// TwinCAT 3 PLC project MAS418_PLC
// ProgramVersion: 3.1.4023.0
// libraries:
//   Tc2_Standard, * (Beckhoff Automation GmbH)
//   Tc2_System, * (Beckhoff Automation GmbH)
//   Tc3_Module, * (Beckhoff Automation GmbH)
//   VisuSymbols,3.5.10.0,System
// project tree:
//   / GlobalTextList.TcGTLO, PlcTask.TcTTO, Visualization Manager.TcVMO (not stored)
//   ControlBox/GVLs/ G_Inputs.TcGVL, G_RealControlBox.TcGVL, G_VB.TcGVL
//   ControlBox/POUs/FunctionBlocks/ FB_ModeRealControlBox.TcPOU, FB_ModeSelector.TcPOU, FB_ModeVisualControlBox.TcPOU (not stored)
//   ControlBox/VISUs/ V_VB.TcVIS
//   Inputs/FunctionBlocks/ FB_AnalogInputScaling.TcPOU, FB_Encoder.TcPOU, FB_FlowMeterInputScaling.TcPOU, FB_JoystickInputScaling.TcPOU
//   Inputs/GVLs/ G_ScaledSensorData.TcGVL, G_RawSensorData.TcGVL
//   Inputs/ P_Inputs.TcPOU
//   Inputs/Structs/ ST_AnalogInput.TcDUT, ST_AnalogInputScaling.TcDUT, ST_AnalogInputStatus.TcDUT, ST_FlowMeterInputScaling.TcDUT, ST_JoystickInputScaling.TcDUT
//   MotionControl/DUTs/ ST_OpenLoopControlCylinderSettings.TcDUT, ST_OpenLoopControlWinchSettings.TcDUT, ST_Parameters.TcDUT, ST_ValveOutput.TcDUT, ST_ValveDeadBand.TcDUT
//   MotionControl/FunctionBlocks/MainBlocks/ FB_ManualControl.TcPOU
//   MotionControl/FunctionBlocks/SubBlocks/ FB_Joystick.TcPOU, FB_OpenLoopCylinderControl.TcPOU, FB_OpenLoopWinchControl.TcPOU, FB_ValveOutput.TcPOU
//   MotionControl/GVLs/ G_Outputs.TcGVL, G_Parameters.TcGVL, G_Work.TcGVL
//   MotionControl/POUs/ P_CraneControl.TcPOU, P_Outputs.TcPOU
//   Programs/ MAIN.TcPOU
//   ControlBox/DUTs/ E_Button.TcDUT (not stored), E_Joy.TcDUT (not stored), E_Light.TcDUT (not stored), E_Mode.TcDUT, E_Status.TcDUT (not stored)
//   ControlBox/Interfaces/ I_ControlType.TcIO, I_Mode.TcIO (not stored)
// real-time tasks:
//   TASK PlcTask: cycle T#10ms, priority 20, ADS port 350
// I/O:
//   DEVICE Device 4 (EtherCAT) (disabled), AmsNetId 5.80.90.242.5.1
//     Term 1 (EK1100) [EK1100 EtherCAT Coupler (2A E-Bus)]
//       Term 2 (EL1008)
//       Term 3 (EL2008)
//       Term 4 (EL3068)
//       Term 5 (EL3068)
//       Term 6 (EL3174) [EL3174 4Ch. Ana. Input +/-10V Diff., +/-20mA SingleEnded, 16 Bit]
//       Term 7 (EL3255)
//       Term 8 (EL4104)
//       Term 10 (EL9011) [EL9011 End Terminal]
//     Box 9 (Fraba EtherCAT) [Absolute Rotary Encoder IXARC V01.05]
// variable links:
//   MAS418-PLC/MAS418-PLC Instance <-> Device 4 (EtherCAT)/Term 1 (EK1100)/Term 2 (EL1008)
//     PlcTask Inputs/G_RawSensorData.bAutoModeSelector <-> Channel 2/Input
//     PlcTask Inputs/G_RawSensorData.bJoystickEnable <-> Channel 5/Input
//     PlcTask Inputs/G_RawSensorData.bManualModeSelector <-> Channel 1/Input
//     PlcTask Inputs/G_RawSensorData.bStartButton <-> Channel 3/Input
//     PlcTask Inputs/G_RawSensorData.bStopButton <-> Channel 4/Input
//   MAS418-PLC/MAS418-PLC Instance <-> Device 4 (EtherCAT)/Term 1 (EK1100)/Term 7 (EL3255)
//     PlcTask Inputs/G_RawSensorData.stJoyX.nValue <-> AI Standard Channel 2/Value
//     PlcTask Inputs/G_RawSensorData.stJoyY.nValue <-> AI Standard Channel 3/Value
//     PlcTask Inputs/G_RawSensorData.stPositionCylinder.nValue <-> AI Standard Channel 1/Value

CONFIGURATION MAS418_PLC
    RESOURCE PLC ON TwinCAT3
        TASK PlcTask(INTERVAL := T#10ms, PRIORITY := 20);
        PROGRAM MAIN WITH PlcTask : MAIN;
    END_RESOURCE
END_CONFIGURATION

// ---- Inputs/Structs/ST_AnalogInput.TcDUT
TYPE ST_AnalogInput :
STRUCT
	stStatus AT %I* : ST_AnalogInputStatus;
	nValue AT %I* : INT;
END_STRUCT
END_TYPE

// ---- Inputs/Structs/ST_AnalogInputScaling.TcDUT
TYPE ST_AnalogInputScaling :
STRUCT
	fMaxInputValue : LREAL;
	fMinInputValue : LREAL;
	fMaxOutputValue : LREAL;
	fMinOutputValue : LREAL;
END_STRUCT
END_TYPE

// ---- Inputs/Structs/ST_AnalogInputStatus.TcDUT
TYPE ST_AnalogInputStatus :
STRUCT
	Underrange : BIT;
	Overrange : BIT;
	Limit_1_0 : BIT;
	Limit_1_1 : BIT;
	Limit_2_0 : BIT;
	Limit_2_1 : BIT;
	Error : BIT;
	Reserved_0_7 : BIT;
	Reserved_1_0 : BIT;	
	Reserved_1_1 : BIT;
	Reserved_1_2 : BIT;	
	Reserved_1_3 : BIT;		
	Reserved_1_4 : BIT;	
	Reserved_1_5 : BIT;	
	TxPDO_State : BIT;
	TxPDO_Toggle : BIT;
END_STRUCT
END_TYPE

// ---- Inputs/Structs/ST_FlowMeterInputScaling.TcDUT
TYPE ST_FlowMeterInputScaling :
STRUCT
	fMaxInputValue : LREAL;
	fMinInputValue : LREAL;
	fNeutralInputValue : LREAL;
	fNeutralDeadband : LREAL;
	fMaxOutputValue : LREAL;
	fMinOutputValue : LREAL;
	fNeutralOutputValue : LREAL;
END_STRUCT
END_TYPE

// ---- Inputs/Structs/ST_JoystickInputScaling.TcDUT
TYPE ST_JoystickInputScaling :
STRUCT
	fMaxInputValue : LREAL;
	fMinInputValue : LREAL;
	fNeutralInputValue : LREAL;
	fNeutralDeadband : LREAL;
	fMaxOutputValue : LREAL;
	fMinOutputValue : LREAL;
	fNeutralOutputValue : LREAL;
END_STRUCT
END_TYPE

// ---- MotionControl/DUTs/ST_OpenLoopControlCylinderSettings.TcDUT
TYPE ST_OpenLoopControlCylinderSettings :
STRUCT
	fBoreArea : LREAL := 0.0033183;
	fAnnulusArea : LREAL := 0.0023562;
	fMaxFlowCapacity : LREAL := 75;
END_STRUCT
END_TYPE

// ---- MotionControl/DUTs/ST_OpenLoopControlWinchSettings.TcDUT
TYPE ST_OpenLoopControlWinchSettings :
STRUCT
	fWichDrumDiameter : LREAL := 0.0475;
	fWinchDisplacement : LREAL := 32;
	fGearBox : LREAL := 20;
	fMaxFlow : LREAL := 60;
	fWinchDrumScaling : LREAL := 0.000744309;
END_STRUCT
END_TYPE

// ---- MotionControl/DUTs/ST_Parameters.TcDUT
TYPE ST_Parameters :
STRUCT
	fCyclicTime : LREAL := 0.01;
	fMaxVelocityLimit : LREAL := 0.05;
	stOpenLoopControlCylinderSettings : ST_OpenLoopControlCylinderSettings;
	stOpenLoopControlWinchSettings : ST_OpenLoopControlWinchSettings;
	fEncoderOffset : LREAL := 17574.8; 
	bDeadBandCompOn : BOOL := TRUE;
	stWinchValveDeadBand : ST_ValveDeadBand := (fPosMax := 29490.0, fPosMin := 20950.0, fNegMin := 18250.0, fNegMax := 9830.0);
	stCylValveDeadBand 	: ST_ValveDeadBand := (fPosMax := 29490.0, fPosMin := 20950.0, fNegMin := 18250.0, fNegMax := 9830.0);
	stJoystickInputScalingY	: ST_JoystickInputScaling := (fMaxInputValue := 20509.0, fMinInputValue := 11787.0, fNeutralInputValue := 16175, fNeutralDeadband := 50.0, fMaxOutputValue := 1.0, fMinOutputValue := -1.0, fNeutralOutputValue := 0.0);
	stJoystickInputScalingX	: ST_JoystickInputScaling := (fMaxInputValue := 20509.0, fMinInputValue := 11787.0, fNeutralInputValue := 16175, fNeutralDeadband := 50.0, fMaxOutputValue := 1.0, fMinOutputValue := -1.0, fNeutralOutputValue := 0.0);
	stCylPistonPositionScaling : ST_AnalogInputScaling := (fMaxInputValue := 32295.0, fMinInputValue := 229.0, fMaxOutputValue := 0.5, fMinOutputValue := 0.0);
	stPressureSensorScaling400bar : ST_AnalogInputScaling := (fMaxInputValue := 32767.0, fMinInputValue := 0.0, fMaxOutputValue := 400.0, fMinOutputValue := 0.0);
	stPressureSensorScaling40bar : ST_AnalogInputScaling := (fMaxInputValue := 32767.0, fMinInputValue := 0.0, fMaxOutputValue := 40.0, fMinOutputValue := 0.0);
	stFlowMeterInputScaling : ST_FlowMeterInputScaling := (fMaxInputValue := 32295.0, fMinInputValue := 0.0, fNeutralInputValue := 15450, fNeutralDeadband := 50.0, fMaxOutputValue := 150.0, fMinOutputValue := -150.0, fNeutralOutputValue := 0.0);
END_STRUCT
END_TYPE

// ---- MotionControl/DUTs/ST_ValveOutput.TcDUT
TYPE ST_ValveOutput :
STRUCT
	bEnable AT %Q* : BOOL := 0;
	nValveOutput AT %Q* : INT := 19660;
END_STRUCT
END_TYPE

// ---- MotionControl/DUTs/ST_ValveDeadBand.TcDUT
TYPE ST_ValveDeadBand :
STRUCT
	fPosMax : LREAL;
	fPosMin : LREAL;
	fNegMin : LREAL;
	fNegMax : LREAL;
END_STRUCT
END_TYPE

// ---- ControlBox/DUTs/E_Mode.TcDUT
TYPE E_Mode :
(
	OFF := 1,
	Manual,
	Auto
)USINT;
END_TYPE

// ---- ControlBox/GVLs/G_Inputs.TcGVL
VAR_GLOBAL
	fJoyX : LREAL;
	fJoyY : LREAL;
	bOff : BOOL;
	bManual : BOOL;
	bAuto : BOOL;
	bStart : BOOL;
	bStop : BOOL;
	bTopSwitch : BOOL;
	bFault : BOOL;
	bConfirmationStop : BOOL;
	bConfirmation : BOOL;
END_VAR

// ---- ControlBox/GVLs/G_RealControlBox.TcGVL
{attribute 'qualified_only'}
VAR_GLOBAL
END_VAR

// ---- ControlBox/GVLs/G_VB.TcGVL
{attribute 'qualified_only'}
VAR_GLOBAL
	eMode : E_Mode;
	eStatus : E_Status;
	bOn : BOOL := FALSE;
	bAuto : BOOL;
	bStart : BOOL;
	bStop : BOOL;
	bRunning : BOOL;
	bConfirmation : BOOL;
	bConfirmationStop : BOOL;
	bTopSwitch : BOOL;
	bFault : BOOL;
	fJoyY : LREAL;
	fJoyX : LREAL;
END_VAR

// ---- Inputs/GVLs/G_ScaledSensorData.TcGVL
{attribute 'qualified_only'}
VAR_GLOBAL
	fJoystickNormalizedY : LREAL;
	fJoystickNormalizedX : LREAL;
	fPositionCylPiston : LREAL;
	fPressureSupply : LREAL; 
	fPressureReturn : LREAL;
	fPressureCyl_A_PistonSide : LREAL;
	fPressureCyl_B_RodSide : LREAL; 
	fPressureWinch_A_Input : LREAL;
	fPressureWinch_A1_Input : LREAL;
	fPressureWinch_B_Output : LREAL;
	fPressureWinch_B1_Output : LREAL;
	fPressureWinchDrain : LREAL;
	fWinchEncoderPosition : LREAL;
	fWinchWirePosition : LREAL;
	fWinchFlow : LREAL;
END_VAR

// ---- MotionControl/GVLs/G_Outputs.TcGVL
{attribute 'qualified_only'}
VAR_GLOBAL
	bGreenLED AT %Q* : BOOL;
	bRedLED AT %Q* : BOOL;
	
	stWinchValveOutput : ST_ValveOutput;
	stCylValveOutput : ST_ValveOutput;
END_VAR

// ---- MotionControl/GVLs/G_Parameters.TcGVL
{attribute 'qualified_only'}
VAR_GLOBAL
END_VAR

// ---- MotionControl/GVLs/G_Work.TcGVL
{attribute 'qualified_only'}
VAR_GLOBAL
	bManualMode : BOOL;
	bAutoMode : BOOL;
	bWinchEnable : BOOL;
	bCylEnable : BOOL;
	fWinchControlInput : LREAL; 
	fWinchTime : LREAL;
	fCylControlInput : LREAL;
	fCylTime : LREAL;
	fVelRefWinch : LREAL;
	fPosRefWinch : LREAL;
	fControlSignWinch : LREAL;
END_VAR

// ---- Inputs/GVLs/G_RawSensorData.TcGVL
{attribute 'qualified_only'}
VAR_GLOBAL
	bManualModeSelector	AT %I* : BOOL;
	bAutoModeSelector AT %I* : BOOL;
	bOffModeSelector AT %I* : BOOL;
	bStartButton AT %I* : BOOL;
	bStopButton AT %I* : BOOL;
	bJoystickEnable AT %I* : BOOL;
	fFlowWinch AT %I* : LREAL;
	
	
	stJoyX : ST_AnalogInput;
	stJoyY : ST_AnalogInput;
	stPositionCylinder : ST_AnalogInput;
	nEncoderValue AT %I* : UDINT;
	
	stPressureSupply : ST_AnalogInput;
 	stPressureReturn : ST_AnalogInput;
	stPressureCyl_A_PistonSide : ST_AnalogInput;
	stPressureCyl_B_RodSide : ST_AnalogInput;
	stPressureWinch_A_Input : ST_AnalogInput;
	stPressureWinch_A1_Input : ST_AnalogInput;
	stPressureWinch_B_Output : ST_AnalogInput;
	stPressureWinch_B1_Output : ST_AnalogInput;
	stPressureWinchDrain : ST_AnalogInput;
	
	stFlowWinch : ST_AnalogInput; 
END_VAR

// ---- ControlBox/Interfaces/I_ControlType.TcIO
INTERFACE I_ControlType

METHOD Joystick
VAR_INPUT
	bSwitch : BOOL;
	bActive : BOOL;
END_VAR
END_METHOD

METHOD Mode
VAR_INPUT
	eCurrentMode : E_Mode;
END_VAR
END_METHOD

METHOD Status
VAR_INPUT
	eStatus : E_Status;
END_VAR
END_METHOD

END_INTERFACE

// ---- Programs/MAIN.TcPOU
PROGRAM MAIN
VAR
	fbModeSelector : FB_ModeSelector;	
	
END_VAR

fbModeSelector(bControlBox := TRUE);
P_CraneControl();
P_Inputs();
P_Outputs();

END_PROGRAM

// ---- ControlBox/POUs/FunctionBlocks/FB_ModeSelector.TcPOU
FUNCTION_BLOCK FB_ModeSelector
VAR_INPUT
	bControlBox : BOOL;
END_VAR
VAR_OUTPUT
END_VAR
VAR
	fbModeRealControlBox : FB_ModeRealControlBox;
	fbModeVisualControlBox : FB_ModeVisualControlBox;
	fbMode : I_ControlType := fbModeVisualControlBox;
END_VAR

IF NOT(bControlBox) THEN
	fbMode := fbModeVisualControlBox;
		IF (G_VB.bFault) THEN
			fbMode.Mode(E_Mode.OFF);
			fbMode.Status(E_Status.Fault);
			fbMode.Joystick(bActive := FALSE, bSwitch := FALSE);
		ELSE
			IF NOT(G_VB.bOn) THEN
				fbMode.Mode(E_Mode.OFF);
				fbMode.Status(E_Status.NotReady);
				fbMode.Joystick(bActive := FALSE, bSwitch := FALSE);
			ELSIF (G_VB.bOn) AND (G_VB.bAuto) THEN
				fbMode.Mode(E_Mode.Auto);
				fbMode.Joystick(bActive := FALSE, bSwitch := FALSE);
					IF (G_VB.bStop) AND NOT(G_VB.bConfirmationStop) THEN
						fbMode.Status(E_Status.Stoping);
					ELSIF (G_VB.bStart) AND NOT(G_VB.bConfirmation) AND NOT(G_VB.bStop) THEN
						fbMode.Status(E_Status.Starting);
					ELSIF (G_VB.bStart) AND (G_VB.bConfirmation) AND NOT(G_VB.bStop) THEN
						fbMode.Status(E_Status.Running);
					ELSE
						fbMode.Status(E_Status.Ready);
					END_IF
			ELSIF (G_VB.bOn) AND NOT(G_VB.bAuto) THEN
				fbMode.Mode(E_Mode.Manual);
					IF (G_VB.bStop) AND NOT(G_VB.bConfirmationStop) THEN
						fbMode.Status(E_Status.Stoping);
						fbMode.Joystick(bActive := FALSE, bSwitch := FALSE);
					ELSIF (G_VB.bStart) AND NOT(G_VB.bConfirmation) AND NOT(G_VB.bStop) THEN
						fbMode.Status(E_Status.Starting);
						fbMode.Joystick(bActive := FALSE, bSwitch := FALSE);
					ELSIF (G_VB.bStart) AND (G_VB.bConfirmation) AND NOT(G_VB.bStop) THEN
						fbMode.Status(E_Status.Running);
						IF (G_VB.bTopSwitch) THEN
							fbMode.Joystick(bActive := TRUE, bSwitch := TRUE);
						ELSE
							fbMode.Joystick(bActive := TRUE, bSwitch := FALSE);
						END_IF
					ELSE
						fbMode.Status(E_Status.Ready);
						fbMode.Joystick(bActive := FALSE, bSwitch := FALSE);
					END_IF
			END_IF
		END_IF
		
ELSIF (bControlBox) THEN
	fbMode := fbModeRealControlBox;
		IF (G_Inputs.bFault) THEN
			fbMode.Mode(E_Mode.OFF);
			fbMode.Status(E_Status.Fault);
			fbMode.Joystick(bActive := FALSE, bSwitch := FALSE);
		ELSE
			IF (G_RawSensorData.bOffModeSelector) THEN
				fbMode.Mode(E_Mode.OFF);
				fbMode.Status(E_Status.NotReady);
				fbMode.Joystick(bActive := FALSE, bSwitch := FALSE);
			ELSIF (G_RawSensorData.bAutoModeSelector) THEN
				fbMode.Mode(E_Mode.Auto);
				fbMode.Joystick(bActive := FALSE, bSwitch := FALSE);
					IF (G_RawSensorData.bStopButton) AND (G_RawSensorData.fFlowWinch > 1.0) AND (G_RawSensorData.fFlowWinch < -1.0) THEN
						fbMode.Status(E_Status.Stoping);
					ELSIF (G_RawSensorData.bStartButton) AND (NOT(G_Outputs.stCylValveOutput.bEnable) OR NOT(G_Outputs.stWinchValveOutput.bEnable)) THEN
						fbMode.Status(E_Status.Starting);
					ELSIF (G_RawSensorData.bStartButton) AND (G_Outputs.stCylValveOutput.bEnable) AND (G_Outputs.stWinchValveOutput.bEnable) THEN
						fbMode.Status(E_Status.Running);
					ELSE
						fbMode.Status(E_Status.Ready);
					END_IF
			ELSIF (G_RawSensorData.bManualModeSelector) THEN
				fbMode.Mode(E_Mode.Manual);
					IF (G_RawSensorData.bStopButton) AND (G_RawSensorData.fFlowWinch > 1.0) AND (G_RawSensorData.fFlowWinch < -1.0) THEN
						fbMode.Status(E_Status.Stoping);
						fbMode.Joystick(bActive := FALSE, bSwitch := FALSE);
					ELSIF (G_RawSensorData.bStartButton) AND (NOT(G_Outputs.stCylValveOutput.bEnable) OR NOT(G_Outputs.stWinchValveOutput.bEnable)) THEN
						fbMode.Status(E_Status.Starting);
						fbMode.Joystick(bActive := FALSE, bSwitch := FALSE);
					ELSIF (G_RawSensorData.bStartButton) AND (G_Outputs.stCylValveOutput.bEnable) AND (G_Outputs.stWinchValveOutput.bEnable) THEN
						fbMode.Status(E_Status.Running);
						IF (G_RawSensorData.bJoystickEnable) THEN
							fbMode.Joystick(bActive := TRUE, bSwitch := TRUE);
						ELSE
							fbMode.Joystick(bActive := TRUE, bSwitch := FALSE);
						END_IF
					ELSE
						fbMode.Status(E_Status.Ready);
						fbMode.Joystick(bActive := FALSE, bSwitch := FALSE);
					END_IF
			END_IF
		END_IF
END_IF

END_FUNCTION_BLOCK

// ---- ControlBox/POUs/FunctionBlocks/FB_ModeRealControlBox.TcPOU
FUNCTION_BLOCK FB_ModeRealControlBox IMPLEMENTS I_ControlType
VAR_INPUT
END_VAR
VAR_OUTPUT
END_VAR
VAR
END_VAR

METHOD Joystick
VAR_INPUT
	bSwitch	: BOOL;
	bActive : BOOL;
END_VAR
IF NOT(bActive) THEN
	G_Inputs.fJoyY := 0.0;
	G_Inputs.fJoyX := 0.0;
	G_VB.fJoyX := 0.0;
	G_VB.fJoyY := 0.0;
ELSIF (bSwitch) THEN
	G_Inputs.fJoyY := G_VB.fJoyY;
	G_Inputs.fJoyX := 0.0;
	G_VB.fJoyX := 0.0;
ELSIF NOT(bSwitch) THEN
	G_Inputs.fJoyY := 0.0;
	G_Inputs.fJoyX := G_VB.fJoyX;
	G_VB.fJoyY := 0.0;
END_IF
END_METHOD

METHOD Mode
VAR_INPUT
	eCurrentMode : E_Mode;
END_VAR
G_VB.eMode := eCurrentMode;
END_METHOD

METHOD Status
VAR_INPUT
	eStatus : E_Status;
END_VAR
G_VB.eStatus := eStatus;
END_METHOD

END_FUNCTION_BLOCK

// ---- MotionControl/POUs/P_CraneControl.TcPOU
PROGRAM P_CraneControl
VAR
	fbManualControl : FB_ManualControl;
	bEnableManualControl : BOOL;
	fControlOutputNormalizedCylinder : LREAL;
	fControlOutputNormalizedWinch : LREAL;	
END_VAR

fbManualControl(
	eMode := G_VB.eMode,
	eStatus := G_VB.eStatus,
	stParam := G_Parameters.stParam,
);

IF (G_VB.eMode = E_Mode.Manual) AND (G_VB.eStatus = E_Status.Running) THEN
	fControlOutputNormalizedCylinder := LIMIT(-1.0, fbManualControl.fControlOutputNormalizedCylinder, 1.0);
	fControlOutputNormalizedWinch := LIMIT(-1.0, fbManualControl.fControlOutputNormalizedWinch, 1.0);
ELSE
	fControlOutputNormalizedCylinder := 0.0;
	fControlOutputNormalizedWinch := 0.0;
END_IF

G_Work.fWinchControlInput := fControlOutputNormalizedWinch;
G_Work.fCylControlInput := fControlOutputNormalizedCylinder;

END_PROGRAM

// ---- MotionControl/FunctionBlocks/MainBlocks/FB_ManualControl.TcPOU
FUNCTION_BLOCK FB_ManualControl
VAR_INPUT
	eMode : E_Mode;
	eStatus : E_Status;
	stParam : ST_Parameters;
END_VAR
VAR_OUTPUT
	fControlOutputNormalizedCylinder : LREAL;
	fControlOutputNormalizedWinch : LREAL;
END_VAR
	
VAR
	fbJoystick : FB_Joystick;
	fbOpenLoopCylindeControl : FB_OpenLoopCylinderControl;
	fbOpenLoopWinchControl : FB_OpenLoopWinchControl;
END_VAR

IF NOT(G_RawSensorData.bJoystickEnable) THEN
	fbJoystick(
		bEnable := (eMode = E_Mode.Manual),
		stParam := stParam,
		fNormalizedInput := G_ScaledSensorData.fJoystickNormalizedX,
	);
	
	fbOpenLoopCylindeControl(
		bEnable := (eMode = E_Mode.Manual),
		stParam := stParam,
		fInput_ms := fbJoystick.fOutput,
		fNormalizedOutput => fControlOutputNormalizedCylinder,
	);
	
	fbOpenLoopWinchControl(
		bEnable := (eMode = E_Mode.Manual),
		stParam := stParam,
		fInput_ms := 0.0,
		fNormalizedOutput => fControlOutputNormalizedWinch,
	);
	
ELSIF	(G_RawSensorData.bJoystickEnable) THEN
	fbJoystick(
		bEnable := (eMode = E_Mode.Manual),
		stParam := stParam,
		fNormalizedInput := G_ScaledSensorData.fJoystickNormalizedY
	);
	
	fbOpenLoopCylindeControl(
		bEnable := (eMode = E_Mode.Manual),
		stParam := stParam,
		fInput_ms := 0.0,
		fNormalizedOutput => fControlOutputNormalizedCylinder,
	);
	
	fbOpenLoopWinchControl(
		bEnable := (eMode = E_Mode.Manual),
		stParam := stParam,
		fInput_ms := fbJoystick.fOutput,
		fNormalizedOutput => fControlOutputNormalizedWinch,
	);
END_IF

END_FUNCTION_BLOCK

// ---- MotionControl/FunctionBlocks/SubBlocks/FB_Joystick.TcPOU
FUNCTION_BLOCK FB_Joystick
VAR_INPUT
	bEnable : BOOL;
	fNormalizedInput : LREAL;
	stParam : ST_Parameters;
END_VAR
VAR_OUTPUT
	fOutput : LREAL;
END_VAR
VAR
END_VAR

IF (bEnable) THEN
	fOutput := fNormalizedInput*G_Parameters.stParam.fMaxVelocityLimit;
ELSE
	fOutput := 0.0;
END_IF

END_FUNCTION_BLOCK

// ---- MotionControl/FunctionBlocks/SubBlocks/FB_OpenLoopCylinderControl.TcPOU
FUNCTION_BLOCK FB_OpenLoopCylinderControl
VAR_INPUT
	bEnable : BOOL;
	fInput_ms : LREAL;
	stParam : ST_Parameters;
END_VAR
VAR_OUTPUT
	fNormalizedOutput : LREAL;
END_VAR
VAR
	fFlowReference_m3s : LREAL; 
	fM3sToLmin : LREAL := 60000;
END_VAR

IF (fInput_ms >= 0.0) THEN
	fFlowReference_m3s := stParam.stOpenLoopControlCylinderSettings.fBoreArea * fInput_ms;
ELSE
	fFlowReference_m3s := fInput_ms * stParam.stOpenLoopControlCylinderSettings.fAnnulusArea;
END_IF

IF (bEnable) THEN
	fNormalizedOutput := (fM3sToLmin * fFlowReference_m3s) / stParam.stOpenLoopControlCylinderSettings.fMaxFlowCapacity;
ELSE
	fNormalizedOutput := 0.0;
END_IF

IF (fNormalizedOutput > 1.0) THEN
	fNormalizedOutput := 1.0;
ELSIF (fNormalizedOutput < -1.0) THEN
	fNormalizedOutput := -1.0;
END_IF;

END_FUNCTION_BLOCK

// ---- MotionControl/FunctionBlocks/SubBlocks/FB_OpenLoopWinchControl.TcPOU
FUNCTION_BLOCK FB_OpenLoopWinchControl
VAR_INPUT
	bEnable : BOOL; 
	FInput_ms : LREAL;
	stParam : ST_Parameters; 
END_VAR
VAR_OUTPUT
	fNormalizedOutput : LREAL;
END_VAR
VAR
	fFlowReference_m3s : LREAL;
	fM3sToLmin : LREAL := 60000;
END_VAR

fFlowReference_m3s := stParam.stOpenLoopControlWinchSettings.fWinchDisplacement * 1000000 * fInput_ms / stParam.stOpenLoopControlWinchSettings.fGearBox;


IF (bEnable) THEN
	fNormalizedOutput := (fM3sToLmin * fFlowReference_m3s) / stParam.stOpenLoopControlWinchSettings.fMaxFlow;
ELSE
	fNormalizedOutput := 0.0;
END_IF

IF (fNormalizedOutput > 1.0) THEN
	fNormalizedOutput := 1.0;
ELSIF (fNormalizedOutput < -1.0) THEN
	fNormalizedOutput := -1.0;
END_IF;

END_FUNCTION_BLOCK

// ---- Inputs/P_Inputs.TcPOU
PROGRAM P_Inputs
VAR
	fbJoystickWinch	: FB_JoystickInputScaling;
	fbJoystickCyl : FB_JoystickInputScaling;
	fbWinchPosition : FB_Encoder;
	fbCylPistonPosition : FB_AnalogInputScaling;
	fbPressureSupply : FB_AnalogInputScaling;
	fbPressureReturn : FB_AnalogInputScaling;
	fbPressureCyl_A_PistonSide : FB_AnalogInputScaling;
	fbPressureCyl_B_RodSide : FB_AnalogInputScaling;
	fbPressureWinch_A_Input : FB_AnalogInputScaling;
	fbPressureWinch_A1_Input : FB_AnalogInputScaling;
	fbPressureWinch_B_Output : FB_AnalogInputScaling;
	fbPressureWinch_B1_Output : FB_AnalogInputScaling;
	fbPressureWinchDrain : FB_AnalogInputScaling;
	fbFlowWinch : FB_FlowMeterInputScaling;
END_VAR

fbJoystickWinch(
	bEnable := G_RawSensorData.bManualModeSelector,
	nRawInput := G_RawSensorData.stJoyY.nValue,
	stJoystickInputScaling := G_Parameters.stParam.stJoystickInputScalingY,
	fNormalizedOutput => G_ScaledSensorData.fJoystickNormalizedY
);
fbJoystickCyl(
	bEnable := G_RawSensorData.bManualModeSelector,
	nRawInput := G_RawSensorData.stJoyX.nValue,
	stJoystickInputScaling := G_Parameters.stParam.stJoystickInputScalingX,
	fNormalizedOutput => G_ScaledSensorData.fJoystickNormalizedX
);
fbWinchPosition (
nRawInput := G_RawSensorData.nEncoderValue, 
fPosition => G_ScaledSensorData.fWinchEncoderPosition,
);
G_ScaledSensorData.fWinchWirePosition := fbWinchPosition.fPosition*G_Parameters.stParam.stOpenLoopControlWinchSettings.fWinchDrumScaling;
fbCylPistonPosition(
	nRawInput := G_RawSensorData.stPositionCylinder.nValue,
	stAnalogInputScaling := G_Parameters.stParam.stCylPistonPositionScaling,
	fOutput => G_ScaledSensorData.fPositionCylPiston
);
fbPressureSupply(
	nRawInput := G_RawSensorData.stPressureSupply.nValue,
	stAnalogInputScaling := G_Parameters.stParam.stPressureSensorScaling400bar,
	fOutput => G_ScaledSensorData.fPressureSupply
);
fbPressureReturn(
	nRawInput := G_RawSensorData.stPressureReturn.nValue,
	stAnalogInputScaling := G_Parameters.stParam.stPressureSensorScaling40bar,
	fOutput => G_ScaledSensorData.fPressureReturn
);
fbPressureCyl_A_PistonSide(
	nRawInput := G_RawSensorData.stPressureCyl_A_PistonSide.nValue,
	stAnalogInputScaling := G_Parameters.stParam.stPressureSensorScaling400bar,
	fOutput => G_ScaledSensorData.fPressureCyl_A_PistonSide
);
fbPressureCyl_B_RodSide(
	nRawInput := G_RawSensorData.stPressureCyl_B_RodSide.nValue,
	stAnalogInputScaling := G_Parameters.stParam.stPressureSensorScaling400bar,
	fOutput => G_ScaledSensorData.fPressureCyl_B_RodSide
);
fbPressureWinch_A_Input(
	nRawInput := G_RawSensorData.stPressureWinch_A_Input.nValue,
	stAnalogInputScaling := G_Parameters.stParam.stPressureSensorScaling400bar,
	fOutput => G_ScaledSensorData.fPressureWinch_A_Input
);
fbPressureWinch_A1_Input(
	nRawInput := G_RawSensorData.stPressureWinch_A1_Input.nValue,
	stAnalogInputScaling := G_Parameters.stParam.stPressureSensorScaling400bar,
	fOutput => G_ScaledSensorData.fPressureWinch_A1_Input
);
fbPressureWinch_B_Output(
	nRawInput := G_RawSensorData.stPressureWinch_B_Output.nValue,
	stAnalogInputScaling := G_Parameters.stParam.stPressureSensorScaling400bar,
	fOutput => G_ScaledSensorData.fPressureWinch_B_Output
);
fbPressureWinch_B1_Output(
	nRawInput := G_RawSensorData.stPressureWinch_B1_Output.nValue,
	stAnalogInputScaling := G_Parameters.stParam.stPressureSensorScaling400bar,
	fOutput => G_ScaledSensorData.fPressureWinch_B1_Output
);
fbPressureWinchDrain(
	nRawInput := G_RawSensorData.stPressureWinchDrain.nValue,
	stAnalogInputScaling := G_Parameters.stParam.stPressureSensorScaling40bar,
	fOutput => G_ScaledSensorData.fPressureWinchDrain
);
fbFlowWinch(
	nRawInput := G_RawSensorData.stFlowWinch.nValue,
	stFlowMeterInputScaling := G_Parameters.stParam.stFlowMeterInputScaling,
	fNormalizedOutput => G_ScaledSensorData.fWinchFlow
);

END_PROGRAM

// ---- Inputs/FunctionBlocks/FB_JoystickInputScaling.TcPOU
FUNCTION_BLOCK FB_JoystickInputScaling
VAR_INPUT
	bEnable : BOOL;
	nRawInput : INT;
	stJoystickInputScaling : ST_JoystickInputScaling;
END_VAR
VAR_OUTPUT
	fNormalizedOutput : LREAL;
END_VAR
VAR
	fRawInput : LREAL;
	fTempInput : LREAL;
	fTempOutput : LREAL;
END_VAR

fRawInput := INT_TO_LREAL(nRawInput);

fTempInput := fRawInput - stJoystickInputScaling.fNeutralInputValue;

IF fTempInput > stJoystickInputScaling.fNeutralDeadband THEN 
	fTempOutput := fTempInput/(stJoystickInputScaling.fMaxInputValue - stJoystickInputScaling.fNeutralInputValue);
ELSIF fTempInput < -stJoystickInputScaling.fNeutralDeadband THEN
	fTempOutput := fTempInput/(stJoystickInputScaling.fNeutralInputValue - stJoystickInputScaling.fMinInputValue);
ELSE
	fTempOutput := 0.0;
END_IF
IF NOT(bEnable) THEN
	fNormalizedOutput := 0.0;
ELSE
	fNormalizedOutput := LIMIT(stJoystickInputScaling.fMinOutputValue, fTempOutput, stJoystickInputScaling.fMaxOutputValue);
END_IF

END_FUNCTION_BLOCK

// ---- Inputs/FunctionBlocks/FB_Encoder.TcPOU
FUNCTION_BLOCK FB_Encoder
VAR_INPUT
	nRawInput : UDINT;
	stParam : ST_Parameters;
END_VAR
VAR_OUTPUT
	fPosition : LREAL;
END_VAR
VAR PERSISTENT
	nRounds : DINT;
	nRawLast : DINT;
END_VAR
VAR
	nInput : DINT;
	nTempInputDiff : DINT;
	nCount : DINT; 
	nMaxValue30bit : DINT := 1073741823;
	nThreshold30bit : DINT := nMaxValue30bit/2;
	fScale6bit : LREAL := 360.0/65525.0;
	fTempPosition : LREAL;
END_VAR

nInput := UDINT_TO_DINT(nRawInput);

nTempInputDiff := nInput - nRawLast;
IF (nTempInputDiff > nThreshold30bit) THEN
	nRounds := nRounds - 1;
END_IF

IF (nTempInputDiff < -nThreshold30bit) THEN 
	nRounds := nRounds + 1;
END_IF

nCount := nInput + nRounds*nMaxValue30bit;

fPosition := DINT_TO_LREAL(nCount)*fScale6bit - stParam.fEncoderOffset;

END_FUNCTION_BLOCK

// ---- Inputs/FunctionBlocks/FB_AnalogInputScaling.TcPOU
FUNCTION_BLOCK FB_AnalogInputScaling
VAR_INPUT
	nRawInput : INT;
	stAnalogInputScaling : ST_AnalogInputScaling;
END_VAR
VAR_OUTPUT
	fOutput : LREAL;
END_VAR
VAR
	fRawInput : LREAL; 
	fNormalizedInput : LREAL;
END_VAR

fRawInput := INT_TO_LREAL(nRawInput);

fNormalizedInput := (fRawInput - stAnalogInputScaling.fMinInputValue) / (stAnalogInputScaling.fMaxInputValue - stAnalogInputScaling.fMinInputValue);

fOutput := LIMIT(stAnalogInputScaling.fMinOutputValue, stAnalogInputScaling.fMinOutputValue + fNormalizedInput*(stAnalogInputScaling.fMaxOutputValue - stAnalogInputScaling.fMinOutputValue), stAnalogInputScaling.fMaxOutputValue);

END_FUNCTION_BLOCK

// ---- Inputs/FunctionBlocks/FB_FlowMeterInputScaling.TcPOU
FUNCTION_BLOCK FB_FlowMeterInputScaling
VAR_INPUT
	nRawInput : INT; 
	stFlowMeterInputScaling : ST_FlowMeterInputScaling;
END_VAR
VAR_OUTPUT
	fNormalizedOutput : LREAL;
END_VAR
VAR
	fRawInput : LREAL; 
	fTempInput : LREAL; 
	fTempOutput : LREAL;
END_VAR

fRawInput := INT_TO_LREAL(nRawInput);

fTempInput := fRawInput - stFlowMeterInputScaling.fNeutralInputValue;

IF fTempInput > stFlowMeterInputScaling.fNeutralDeadband THEN 
	fTempOutput := fTempInput/(stFlowMeterInputScaling.fMaxInputValue - stFlowMeterInputScaling.fNeutralInputValue);
ELSIF fTempInput < -stFlowMeterInputScaling.fNeutralDeadband THEN
	fTempOutput := fTempInput/(stFlowMeterInputScaling.fNeutralInputValue - stFlowMeterInputScaling.fMinInputValue);
ELSE
	fTempOutput := 0.0;
END_IF

fNormalizedOutput := LIMIT(stFlowMeterInputScaling.fMinOutputValue, fTempOutput*150.0, stFlowMeterInputScaling.fMaxOutputValue);

END_FUNCTION_BLOCK

// ---- MotionControl/POUs/P_Outputs.TcPOU
PROGRAM P_Outputs
VAR
	fbWinchValveOutput : FB_ValveOutput;
	fbCylValveOutput : FB_ValveOutput;
END_VAR

G_Outputs.stWinchValveOutput.bEnable := G_Work.bManualMode; 
fbWinchValveOutput(
	bEnable := G_Work.bWinchEnable,
	bDeadBandCompOn := G_Parameters.stParam.bDeadBandCompOn,
	stValveDeadBand := G_Parameters.stParam.stWinchValveDeadBand,
	fNormalizedInput := G_Work.fWinchControlInput,
	nOutput => G_Outputs.stWinchValveOutput.nValveOutput
);

G_Outputs.stCylValveOutput.bEnable := G_Work.bManualMode;
fbCylValveOutput(
	bEnable := G_Work.bCylEnable OR G_Work.fCylTime > 0.0,
	bDeadBandCompOn := G_Parameters.stParam.bDeadBandCompOn,
	stValveDeadBand := G_Parameters.stParam.stCylValveDeadBand,
	fNormalizedInput := G_Work.fCylControlInput,
	nOutput => G_Outputs.stCylValveOutput.nValveOutput
);

IF (G_VB.eStatus = E_Status.Running) THEN
	G_Outputs.bGreenLED := TRUE;
	G_Outputs.bRedLED := FALSE;
ELSIF (G_VB.eStatus = E_Status.Fault) OR (G_VB.eStatus = E_Status.Stoping) THEN
	G_Outputs.bRedLED := TRUE;
	G_Outputs.bGreenLED := FALSE;
ELSE
	G_Outputs.bRedLED := FALSE;
	G_Outputs.bGreenLED := FALSE;
END_IF

END_PROGRAM

// ---- MotionControl/FunctionBlocks/SubBlocks/FB_ValveOutput.TcPOU
FUNCTION_BLOCK FB_ValveOutput
VAR_INPUT
	bEnable : BOOL;
	bDeadBandCompOn : BOOL;
	stValveDeadband : ST_ValveDeadBand;
	fNormalizedInput : LREAL;
END_VAR
VAR_OUTPUT
	bEnableValveOutput : BOOL;
	nOutput : INT;
END_VAR
VAR
	nOffset : INT := 19660;
	nMaxValue : INT := 29490;
	nMinValue : INT := 9830;
	nTempOutput : INT;
END_VAR

IF	bDeadBandCompOn THEN
	IF fNormalizedInput > 0.0 THEN
		nTempOutput := LREAL_TO_INT(ABS(fNormalizedInput*(stValveDeadBand.fPosMax - stValveDeadBand.fPosMin) + stValveDeadBand.fPosMin));
	ELSIF fNormalizedInput < 0.0 THEN
		nTempOutput := LREAL_TO_INT(ABS(fNormalizedInput*(stValveDeadBand.fNegMax - stValveDeadBand.fNegMin) - stValveDeadBand.fNegMin));
	ELSE
		nTempOutput := nOffset;
	END_IF
ELSE
	IF fNormalizedInput > 0.0 THEN
		nTempOutput := LREAL_TO_INT(ABS(fNormalizedInput*(32767.0 - 19660.0) + 19660.0));
	ELSIF fNormalizedInput < 0.0 THEN
		nTempOutput := LREAL_TO_INT(ABS(fNormalizedInput*(0 - 19660.0) - 19660.0));
	ELSE
		nTempOutput := nOffset;
	END_IF	
END_IF	
IF bEnable THEN
	nOutput := LIMIT(nMinValue, nTempOutput, nMaxValue);
	bEnableValveOutput := TRUE; 
ELSE 	
	nOutput := nOffset;
	bEnableValveOutput := FALSE;	
END_IF

END_FUNCTION_BLOCK

// ---- GlobalTextList.TcGTLO
TEXTLIST GlobalTextList
  649 = '%s'
  584 = 'Auto\tManual'
  81 = 'GroupBox'
  928 = 'Label'
  533 = 'Mode:'
  167 = 'ON\tOFF'
  149 = 'Start'
  393 = 'Status:'
  97 = 'Stop'
  963 = 'x-axis'
  99 = 'X-axis'
  366 = 'Y-axis'
END_TEXTLIST

// ---- ControlBox/VISUs/V_VB.TcVIS
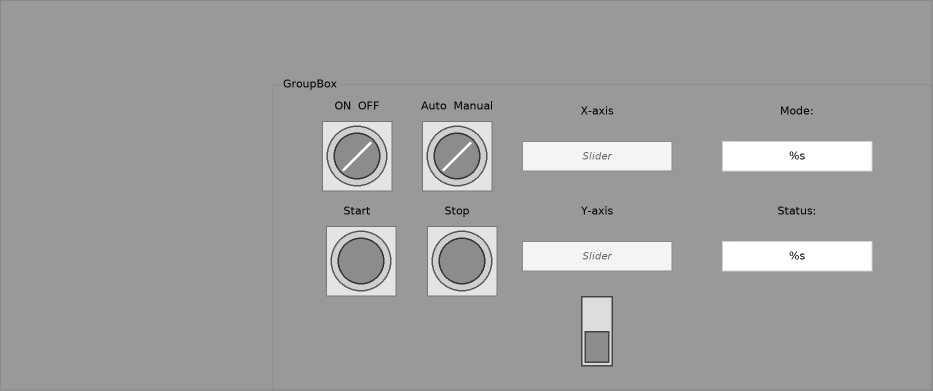
VISUALIZATION V_VB  // 933x391
    GroupBox (272,76 661x315), "GroupBox"
        RotarySwitch (50,45 70x70), variable: G_VB.bOn, behaviour: TOGGLE, style: Switch-RotarySwitch-Gray
        Slider (250,65 150x30), variable: G_VB.fJoyX, scale 0..32767
        Slider (250,165 150x30), variable: G_VB.fJoyY, scale 0..32767
        Label (250,20 150x30), "X-axis"
        Label (250,120 150x30), "Y-axis"
        PushSwitch (54,150 70x70), variable: G_VB.bStart, behaviour: TOGGLE, style: Switch-PushSwitch-Gray
        PushSwitch (155,150 70x70), variable: G_VB.bStop, behaviour: TOGGLE, style: Switch-PushSwitch-Gray
        RotarySwitch (150,45 70x70), variable: G_VB.bAuto, behaviour: TOGGLE, style: Switch-RotarySwitch-Gray
        Label (10,15 150x30), "ON OFF"
        Label (110,15 150x30), "Auto Manual"
        Label (10,120 150x30), "Start"
        Label (110,120 150x30), "Stop"
        DipSwitch (290,220 70x70), variable: G_VB.bTopSwitch, behaviour: TOGGLE, style: Switch-DipSwitch-Gray
        Textfield (450,65 150x30), "%s", text variable: G_VB.eMode
        Textfield (450,165 150x30), "%s", text variable: G_VB.eStatus
        Label (450,20 150x30), "Mode:"
        Label (450,120 150x30), "Status:"
END_VISUALIZATION
